// Helper to generate a message with replaced arguments
FUNCTION F_Print : STRING(255)
VAR_INPUT
    sMessage:				STRING(255);
    sArguments:				STRING(255);	// Arguments are separated by $R 
END_VAR
VAR
    sArg:					STRING; 		// single argument
    nPosition:				INT;         	// Position of the $R delimiter
    nPlaceholder:			INT;         	// Position of the %s placeholder
END_VAR
(*
    Tc3_Event – TwinCAT 3 Event Logging Framework
    Copyright (c) Peter Zerlauth

    This component is provided under a Dual Licensing Model:

    1. GPLv3 Open-Source License
       - Free for personal, educational, and non-commercial use.
       - Commercial use allowed only if the entire application is published
         under GPLv3, including all modifications to this code.
       - Requires full disclosure of source code for derivative works.

    2. Commercial License
       - Required for integration into proprietary or closed-source products.
       - Removes all GPLv3 copyleft obligations.
       - Includes optional warranty, professional support, and long-term
         maintenance options.

    For commercial licensing, contact:
        info@peterzerlauth.com

    By using this Function Block you agree to the terms of the selected license.
*)

// replace placeholders with arguments
F_Print := sMessage;

IF sArguments = '' THEN
    RETURN;
END_IF

nPosition := FIND(sArguments, '$R');
WHILE nPosition > 0 DO
    
    sArg := LEFT(sArguments, nPosition - 1);
    
    nPlaceholder := FIND(F_Print, '%s');
    IF nPlaceholder > 0 THEN
        F_Print := REPLACE(F_Print, sArg, 2, nPlaceholder);
    ELSE
        RETURN;
    END_IF
	
    sArguments := DELETE(sArguments, nPosition, 1);
    nPosition := FIND(sArguments, '$R');
    
END_WHILE

END_FUNCTION

(* stored: Version 1.1.0.1
   POU F_Print: Id {bd1ae1ff-de92-4fbf-9c28-b97df594421e}, SpecialFunc None *)
